// Mitsubishi GX Works2 project: ladder   PLC: FX3U/FX3UC

PROGRAM MAIN
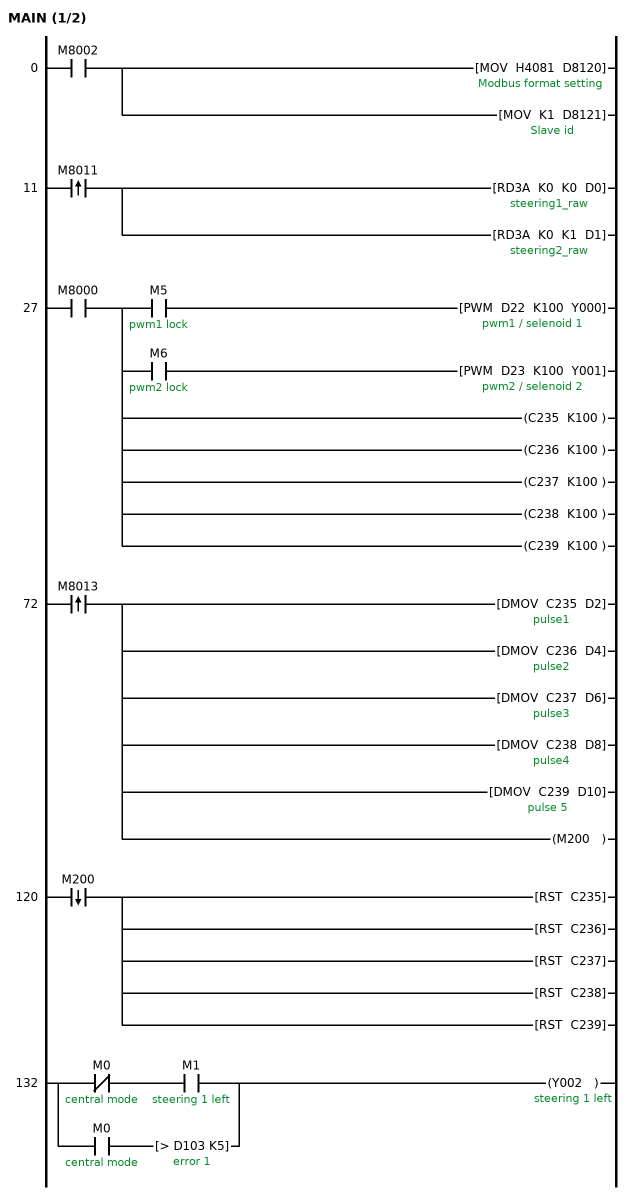
0     LD      M8002
      MOV     H4081 D8120  ; Modbus format setting
      MOV     K1 D8121  ; Slave id
11    LDP     M8011
      RD3A    K0 K0 D0  ; steering1_raw
      RD3A    K0 K1 D1  ; steering2_raw
27    LD      M8000
      MPS
      AND     M5  ; pwm1 lock
      PWM     D22 K100 Y000  ; pwm1 / selenoid 1
      MRD
      AND     M6  ; pwm2 lock
      PWM     D23 K100 Y001  ; pwm2 / selenoid 2
      MPP
      OUT     C235 K100
      OUT     C236 K100
      OUT     C237 K100
      OUT     C238 K100
      OUT     C239 K100
72    LDP     M8013
      DMOV    C235 D2  ; pulse1
      DMOV    C236 D4  ; pulse2
      DMOV    C237 D6  ; pulse3
      DMOV    C238 D8  ; pulse4
      DMOV    C239 D10  ; pulse 5
      OUT     M200
120   LDF     M200
      RST     C235
      RST     C236
      RST     C237
      RST     C238
      RST     C239
132   LDI     M0  ; central mode
      AND     M1  ; steering 1 left
      LD      M0  ; central mode
      AND>    D103 K5  ; error 1
      ORB
      OUT     Y002  ; steering 1 left
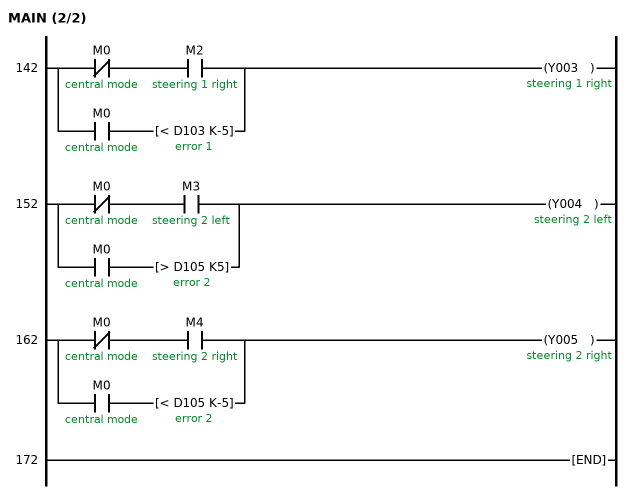
142   LDI     M0  ; central mode
      AND     M2  ; steering 1 right
      LD      M0  ; central mode
      AND<    D103 K-5  ; error 1
      ORB
      OUT     Y003  ; steering 1 right
152   LDI     M0  ; central mode
      AND     M3  ; steering 2 left
      LD      M0  ; central mode
      AND>    D105 K5  ; error 2
      ORB
      OUT     Y004  ; steering 2 left
162   LDI     M0  ; central mode
      AND     M4  ; steering 2 right
      LD      M0  ; central mode
      AND<    D105 K-5  ; error 2
      ORB
      OUT     Y005  ; steering 2 right
172   END
END_PROGRAM

// device comments not shown above
D21  ; steering2_raw
D100  ; steering sensor1
D101  ; steering sensor2
D102  ; setpoint 1
D104  ; setpoint 2
